TEXTLIST TextList_Basiques
  0 = 'OK' | FR: 'OK' | EN: 'OK'
  1 = 'Annul' | FR: 'Annuler' | EN: 'Cancel'
  2 = 'Modifier' | FR: 'Modifier' | EN: 'Modify'
  3 = 'Oui' | FR: 'Oui' | EN: 'Yes'
  4 = 'Non' | FR: 'Non' | EN: 'No'
  5 = 'Créer...' | FR: 'Créer...' | EN: 'Create...'
  6 = 'Modifier...' | FR: 'Modifier...' | EN: 'Modify...'
  7 = 'Supprimer' | FR: 'Supprimer' | EN: 'Delete'
  8 = 'Fermer' | FR: 'Fermer' | EN: 'Close'
  9 = 'Nom' | FR: 'Nom' | EN: 'Name'
  10 = 'Prénom' | FR: 'Prénom' | EN: 'First name'
  11 = 'Créer' | FR: 'Créer' | EN: 'Create'
  12 = 'OPTIONS' | FR: 'OPTIONS' | EN: 'OPTIONS'
  13 = 'Mode_Manuel' | FR: 'Manuel' | EN: 'Manual'
  14 = 'Mode_Auto' | FR: 'Automatique' | EN: 'Automatic'
  15 = 'res' | FR: 'RESET' | EN: 'RESET'
  16 = 'Transfert' | FR: 'Transfert' | EN: 'Transfer'
  17 = 'ch ouvert' | FR: 'Chambre ouverte' | EN: 'Chamber open'
  18 = 'sas ouvert' | FR: 'Sas ouvert' | EN: 'Loadlock open'
  19 = 'modif en ligne' | FR: 'Modification\nen ligne' | EN: 'Online\nmodification'
  22 = 'durée rampe' | FR: 'Durée rampe :' | EN: 'Ramp duration:'
  20 = 'Trac absent' | FR: "ATTENTION : Le logiciel de traçabilité n'est pas lancé! Lancez TrAC" | EN: 'WARNING: Traceability software is not started! Start TrAC'
  21 = 'ACSoft absent' | FR: "ATTENTION : Le logiciel de gestion des évènements n'est pas lancé! Lancez ACSoftware" | EN: 'WARNING: Event logger software is not started! Start ACSoftware'
   = ''
END_TEXTLIST

(* stored: Version 1.1.0.1, ProductVersion 3.1.4024.12
   TextList TextList_Basiques: Id {f858b758-ab46-4477-97dd-d76d30a4cb47} *)
